Fanuc TP program (LS listing): payload.ls

/PROG  PAYLOAD
/ATTR
OWNER		= MNEDITOR;
COMMENT		= "SET PAYLOAD SCH";
PROG_SIZE	= 356;
CREATE		= DATE 23-03-23  TIME 02:24:40;
MODIFIED	= DATE 23-03-23  TIME 02:24:40;
FILE_NAME	= ;
VERSION		= 0;
LINE_COUNT	= 12;
MEMORY_SIZE	= 680;
PROTECT		= READ_WRITE;
TCD:  STACK_SIZE	= 0,
      TASK_PRIORITY	= 50,
      TIME_SLICE	= 0,
      BUSY_LAMP_OFF	= 0,
      ABORT_REQUEST	= 0,
      PAUSE_REQUEST	= 0;
DEFAULT_GROUP	= 1,*,*,*,*;
CONTROL_CODE	= 00000000 00000000;
/APPL
/MN
   1:  IF (DO[174:PART IN T1]=OFF AND DO[175:PART IN T2]=OFF) THEN ;
   2:  PAYLOAD[1:NORMAL WEIGHT] ;
   3:  ENDIF ;
   4:  IF (DO[174:PART IN T1]=ON AND DO[175:PART IN T2]=OFF) THEN ;
   5:  PAYLOAD[2] ;
   6:  ENDIF ;
   7:  IF (DO[174:PART IN T1]=OFF AND DO[175:PART IN T2]=ON) THEN ;
   8:  PAYLOAD[3] ;
   9:  ENDIF ;
  10:  IF (DO[174:PART IN T1]=ON AND DO[175:PART IN T2]=ON) THEN ;
  11:  PAYLOAD[4] ;
  12:  ENDIF ;
/POS
/END
